(* CODESYS project codesys

Project tree, tasks and I/O mapping:
  _750_8216_PFC200 : 750-8212 PFC200, WAGO, order no. 750-8212, version 6.3.1.1
    application Application
      task Task (cyclic, interval t#50ms, priority 15) calls POU
      program MainExtended [ST]
      function block POU_1 [ST]
      program POU [ST]
      program ramita [ST]
    Kbus : Kbus, WAGO, version 2.1.0.1
        unmapped channels: K-BUS diagnostics
    Serial
      COM1 : COM1, WAGO, version 0.0.0.19
    TP600_Onboard_IO : TP600 Onboard IO, WAGO, version 0.0.1.2
        unmapped channels: _IN, _OUT
*)

// _750_8216_PFC200/Application/POU
PROGRAM POU
VAR
	duvan:string;
END_VAR

duvan:='hola';

END_PROGRAM

// _750_8216_PFC200/Application/MainExtended
PROGRAM MainExtended
VAR
END_VAR

END_PROGRAM

// _750_8216_PFC200/Application/POU_1
FUNCTION_BLOCK POU_1
VAR_INPUT
END_VAR
VAR_OUTPUT
END_VAR
VAR
	nuebopou:INT;
END_VAR

END_FUNCTION_BLOCK

// _750_8216_PFC200/Application/ramita
PROGRAM ramita
VAR
	entero:INT;
	
END_VAR

entero:=33;

END_PROGRAM
